FUNCTION_BLOCK AlbertsMachine EXTENDS TcoCore.TcoObject 
VAR
	Automat : AlbertsAutomat(THIS^,eRestoreMode.None);
	Components : AlbertsComponents(THIS^);
	_name :STRING;
	_technologicalDataManager : AlbertsDataManager(THIS^);
END_VAR

Automat.Run();
_technologicalDataManager();

PROPERTY Name : String
GET
END_GET
END_PROPERTY

PROPERTY TechnologicalDataManager : REFERENCE TO AlbertsDataManager
GET
TechnologicalDataManager REF= _technologicalDataManager;
END_GET
END_PROPERTY

END_FUNCTION_BLOCK

(* stored: Version 1.1.0.1, ProductVersion 3.1.4024.5
   POU AlbertsMachine: Id {5b991b17-c4f5-0206-3497-33df35fde26a}, SpecialFunc None
   Property Name: Id {bf1dc4ef-e185-055f-1d35-720b5c79a95e}
   Get Get: Id {34481917-a0c7-0533-1fba-642318e16213}
   Property TechnologicalDataManager: Id {17ae5308-03f2-0215-28b2-6f7448a51b6b}
   Get Get: Id {69297e09-9ee4-09c7-1a1e-5dc766d9637f} *)
